FUNCTION_BLOCK DynamicStringBuffer
VAR_INPUT
END_VAR
VAR_OUTPUT
	Error						:	ST_ERROR;								// Error information of this FB
END_VAR
VAR
	Fifo						:	FB_StringRingBuffer;					// Necessary to buffer log data until it has been written to file.
	MemMan						:	FB_DynMem_Manager;						// Memory manager, required by DynMem_Buffer.
	MemBuf						:	FB_DynMem_Buffer(ipMemMan := MemMan);	// Provides dynamic buffer for Fifo. Is extended automatically if more than the 
																			// default buffer size is needed.
END_VAR
VAR CONSTANT                                                	
	DEFAULT_BUFFER_SIZE 		: UDINT := 1000;							// Default buffer size for FIFO.
END_VAR

METHOD AddLine : BOOL
VAR_INPUT
	Text	:	T_MAXSTRING;	//	Text to be added to the buffer
END_VAR
ResizeFifoBufferIfNecessary();
Fifo.A_AddTail(putValue := CONCAT(Text, '$N'));
END_METHOD

METHOD AddString : BOOL
VAR_INPUT
	Text	:	T_MAXSTRING;	// 	String to be added to the buffer
END_VAR
ResizeFifoBufferIfNecessary();
Fifo.A_AddTail(putValue := Text);
END_METHOD

METHOD PRIVATE AllocateBuffer : BOOL	// Allocates buffer for the Fifo.
VAR_INPUT
END_VAR
MemBuf.CreateBuffer(nSize:=DEFAULT_BUFFER_SIZE*SIZEOF(BYTE), bReset:=TRUE);
Fifo.pBuffer := MemBuf.pBuffer;
Fifo.cbBuffer := DEFAULT_BUFFER_SIZE*SIZEOF(BYTE);
END_METHOD

METHOD FB_exit : BOOL
VAR_INPUT
	bInCopyCode : BOOL; // if TRUE, the exit method is called for exiting an instance that is copied afterwards (online change).
END_VAR
MemBuf.Clear();
END_METHOD

METHOD FB_init : BOOL
VAR_INPUT
	bInitRetains : BOOL; // if TRUE, the retain variables are initialized (warm start / cold start)
	bInCopyCode : BOOL;  // if TRUE, the instance afterwards gets moved into the copy code (online change)
END_VAR
AllocateBuffer();
END_METHOD

METHOD FB_reinit : BOOL
VAR_INPUT
END_VAR
AllocateBuffer();
END_METHOD

METHOD FlushCache : BOOL
VAR_INPUT
END_VAR
Fifo.A_Reset();
END_METHOD

METHOD PersistToFile : BOOL
VAR_INPUT
	FileName			:	T_MAXSTRING;			//	File name including its path
END_VAR
VAR_INST
	state				:	UINT;		
		
	fbFileOpen      	: 	FB_FileOpen;
	fTrigFileOpened		: 	F_TRIG;
	hFile          		: 	UINT;
	               	
	fbFilePuts			:	FB_FilePuts;
	fTrigFilePuts		:	F_TRIG;
	newLogEntry			:	T_MaxString;
	filePutsTriggered	:	BOOL;
	               	
	fbFileClose    	 	: 	FB_FileClose;
	fTrigFileClose		: 	F_TRIG;
	tonTimeout			:	TON;
END_VAR
VAR CONSTANT
	STATE_IDLE							:	UINT	:=	0;
	STATE_OPEN_FILE						:	UINT	:= 	1;
	STATE_GET_STRING_FROM_FIFO		 	:	UINT 	:= 	2;
	STATE_APPEND_DATA_TO_FILE			:	UINT	:= 	3;
	STATE_CLOSE_FILE					:	UINT	:=	4;
	
	NET_ID 				: 	STRING := '';
	TIMEOUT 			: 	TIME := DEFAULT_ADS_TIMEOUT;
END_VAR
// State machine
CASE state OF
	STATE_IDLE:
		IF Fifo.nCount > 0 THEN 
			filePutsTriggered := FALSE;
			state := STATE_OPEN_FILE;
		END_IF
		
	STATE_OPEN_FILE:
		IF fTrigFileOpened.Q THEN state := STATE_GET_STRING_FROM_FIFO; END_IF

	STATE_GET_STRING_FROM_FIFO: 
		IF NOT filePutsTriggered THEN 
			Fifo.A_RemoveHead(getValue => newLogEntry);	
			state := STATE_APPEND_DATA_TO_FILE;
		END_IF			 
		filePutsTriggered := FALSE;
		
	STATE_APPEND_DATA_TO_FILE:
		filePutsTriggered := TRUE;		
		IF fTrigFilePuts.Q THEN 
			IF Fifo.nCount > 0 THEN state := STATE_GET_STRING_FROM_FIFO; 
			ELSE state := STATE_CLOSE_FILE; END_IF
		END_IF
			
	STATE_CLOSE_FILE:
		IF fTrigFileClose.Q THEN state := STATE_IDLE; END_IF
	
END_CASE

// Function blocks used in state machine
fbFileOpen(
	sNetId := NET_ID, sPathName := FileName, nMode := FOPEN_MODEAPPEND OR FOPEN_MODETEXT, 
	ePath := PATH_GENERIC, bExecute := (state = STATE_OPEN_FILE), tTimeout := TIMEOUT,
	hFile => hFile);
fTrigFileOpened(CLK := fbFileOpen.bBusy);

fbFilePuts(
	sNetId := NET_ID, hFile := hFile, sLine := newLogEntry,
	bExecute := (state = STATE_APPEND_DATA_TO_FILE), tTimeout := TIMEOUT);
fTrigFilePuts(CLK := fbFilePuts.bBusy);	

fbFileClose(
	sNetId := NET_ID, hFile := hFile, 
	bExecute := (state = STATE_CLOSE_FILE) OR tonTimeout.Q, tTimeout := TIMEOUT);
fTrigFileClose(CLK := fbFileClose.bBusy);	

// Timeout writing to file => close file
tonTimeout(IN := state <> STATE_IDLE, PT:=TIMEOUT);	
IF tonTimeout.Q THEN state := STATE_IDLE; END_IF

// Error handling
IF fbFileOpen.bError THEN
	Error.Active := TRUE;
	Error.Code := E_ErrorCode.OpeningFileFailed;
	Error.Info := CONCAT('Opening file failed. Error thrown by FB_FileOpen. Consult Beckhoff InfoSys. Internal Error: ', UDINT_TO_STRING(fbFileOpen.nErrId));
ELSIF fbFilePuts.bError THEN
	Error.Active := TRUE;
	Error.Code := E_ErrorCode.WritingToFileFailed;
	Error.Info := CONCAT('Writing to file failed. Error thrown by FB_FilePuts. Consult Beckhoff InfoSys. Internal Error: ', UDINT_TO_STRING(fbFilePuts.nErrId));
ELSIF fbFileClose.bError THEN
	Error.Active := TRUE;
	Error.Code := E_ErrorCode.ClosingFileFailed;
	Error.Info := CONCAT('Closing file failed. Error thrown by FB_FileClose. Consult Beckhoff InfoSys. Internal Error: ', UDINT_TO_STRING(fbFileClose.nErrId));
ELSIF NOT Fifo.bOk AND Fifo.nCount > 0 THEN
	Error.Active := TRUE;
	Error.Code := E_ErrorCode.FifoOverflow;
	Error.Info := 'FIFO overflow. Check if (a) plc has enough free memory and (b) if no message is written each plc cycle';
ELSE
	Error.Active := FALSE;
	Error.Code := E_ErrorCode.None;
	Error.Info := '';
END_IF
END_METHOD

METHOD PopHead : T_MAXSTRING
VAR_INPUT
END_VAR
VAR
	headString	:	T_MAXSTRING;
END_VAR
Fifo.A_RemoveHead(getValue => headString);
PopHead := headString;
END_METHOD

// Resizes the buffer for the FIFO if necessary
METHOD PRIVATE ResizeFifoBufferIfNecessary : BOOL
VAR_INPUT
END_VAR
VAR
	requiredSize : UDINT;
	newSize : DINT;
END_VAR
requiredSize := Fifo.cbSize + MAX_STRING_LENGTH;

IF requiredSize > Fifo.cbBuffer THEN
	MemBuf.Resize(nSize := requiredSize*SIZEOF(BYTE), bPreserve:=TRUE, bReset:=TRUE);
	Fifo.pBuffer := MemBuf.pBuffer;
	Fifo.cbBuffer := requiredSize;
END_IF
END_METHOD

END_FUNCTION_BLOCK

(* stored: Version 1.1.0.1, ProductVersion 3.1.4024.4
   POU DynamicStringBuffer: Id {660876ea-7fc3-4366-aa3c-17474f122e75}, SpecialFunc None
   Method AddLine: Id {40352fe7-a10a-404f-8748-bb98576a3241}
   Method AddString: Id {6405c45a-0cb8-4431-a2bb-9cf39dc1e728}
   Method AllocateBuffer: Id {bc70064d-9855-4df2-8293-04935db0d914}
   Method FB_exit: Id {410b66b7-6428-4a64-9cb8-9b83e356f18f}
   Method FB_init: Id {771f102d-668b-4145-8c28-016b3bbde940}
   Method FB_reinit: Id {03eb2d50-7f23-4ca8-8fa5-9c07e077aa14}
   Method FlushCache: Id {fa7baa03-4401-42cd-8818-9657ae6b0935}
   Method PersistToFile: Id {9df1c79b-f420-4db7-a528-f4f3a2facd9b}
   Method PopHead: Id {1c3e8de3-af72-4def-8aba-61974c7aa041}
   Method ResizeFifoBufferIfNecessary: Id {743741a9-70d0-433f-8900-11f7ea020fe9} *)
